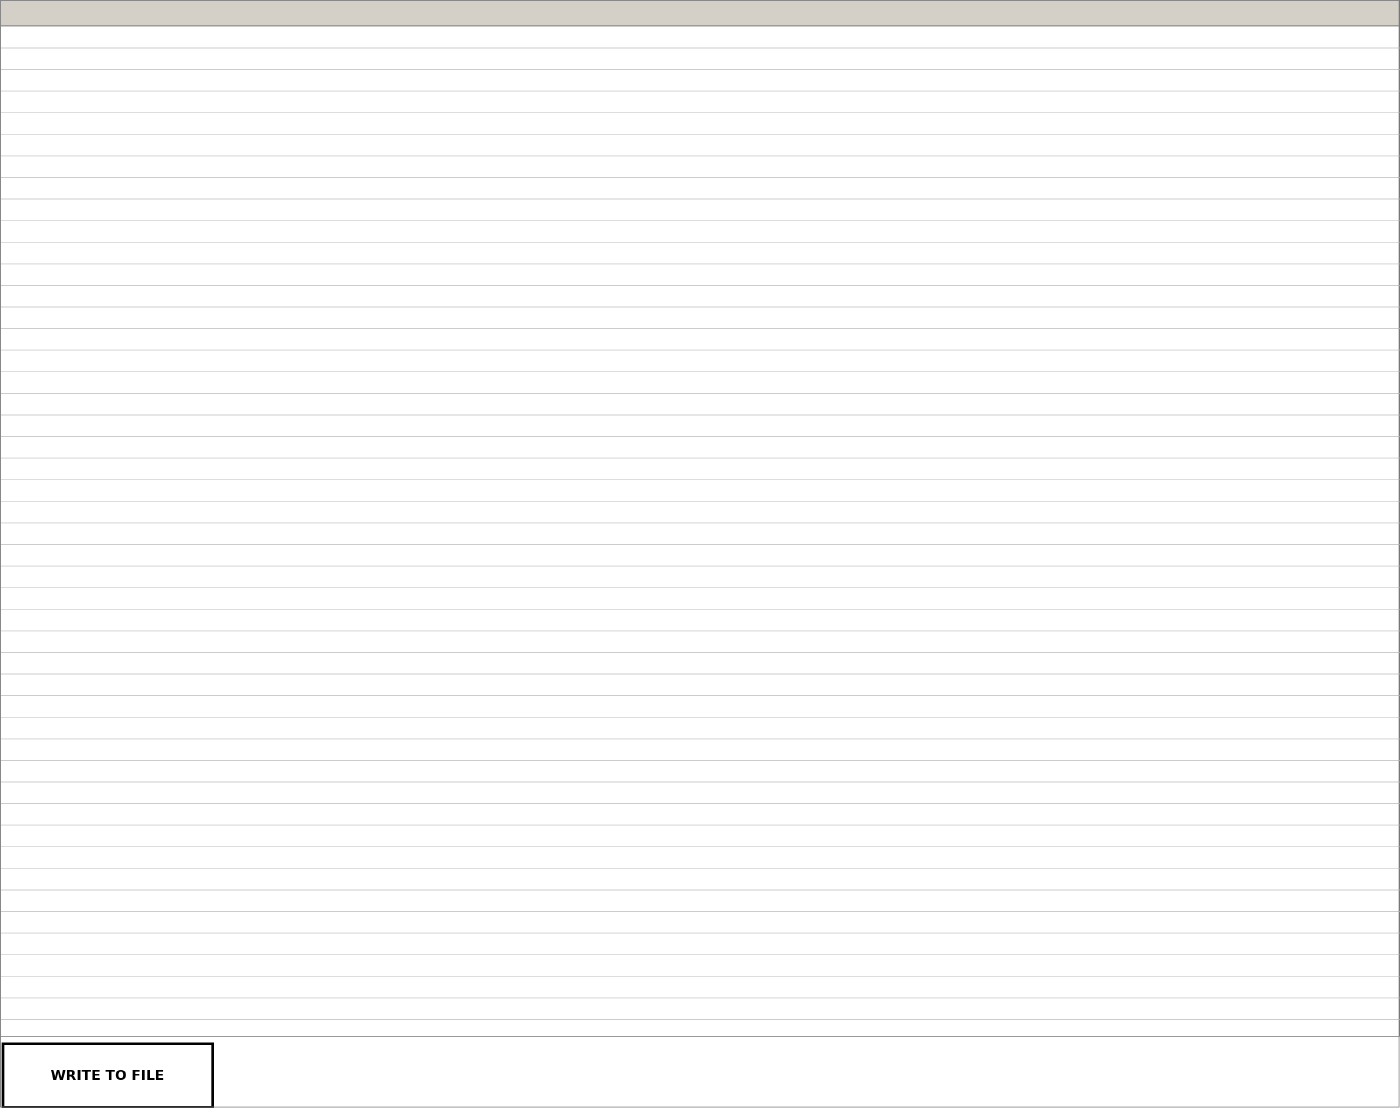
VISUALIZATION Visualization  // 1620x1283
    Table (0,0 1620x1200), data array: MessageData.VisuList
        p1128707560: GVL_AXIS_CTRL.MAX_MESSAGE
        p3854506369: MessageData.VisuList[INDEX].eType
        p1892666644: MessageData.VisuList[INDEX].eDevice
        p338671338: MessageData.VisuList[INDEX].eSubdevice
        p2170511999: MessageData.VisuList[INDEX].iErrorNumber
        p3723444502: MessageData.VisuList[INDEX].tTime
        p1218418051: MessageData.VisuList[INDEX].sText
    Rectangle (2,1207 245x76), "WRITE TO FILE", colour toggle: MAIN.bWriteLog
        toggle MAIN.bWriteLog
END_VISUALIZATION

(* stored: Version 1.1.0.1, ProductVersion 3.1.4024.12
   Visu Visualization: Id {89fb246f-c9b5-08fa-0b54-d9a1901eaa28} *)
